Fanuc TP program (LS listing): approach0.LS

/PROG  approach0
/ATTR
OWNER		= MNEDITOR;
COMMENT		= "test_comment";
PROG_SIZE	= 0;
CREATE		= DATE 31-12-14  TIME 12:00:00;
MODIFIED	= DATE 31-12-14  TIME 12:00:00;
FILE_NAME	= ;
VERSION		= 0;
LINE_COUNT	= 2;
MEMORY_SIZE	= 0;
PROTECT		= READ_WRITE;
TCD:  STACK_SIZE	= 0,
      TASK_PRIORITY	= 50,
      TIME_SLICE	= 0,
      BUSY_LAMP_OFF	= 0,
      ABORT_REQUEST	= 0,
      PAUSE_REQUEST	= 0;
DEFAULT_GROUP	= 1,*,*,*,*,*,*;
CONTROL_CODE	= 00000000 00000000;
/MN
   1:L P[1] 100mm/sec FINE ;
   2:L P[2] 101mm/sec FINE ;
/POS
P[1]{
   GP1:
    UF : 9, UT : 9,
	J1=    0.000 deg,	J2=    0.000 deg,	J3=    0.300 deg,
	J4=    0.600 deg,	J5=    0.500 deg,	J6=    10.000 deg,
	E1=  1000.000  mm,	E2=  1000.000  mm
};
P[2]{
   GP1:
    UF : 9, UT : 9,
	J1=    0.000 deg,	J2=    0.000 deg,	J3=    0.000 deg,
	J4=    0.000 deg,	J5=    0.000 deg,	J6=    0.000 deg,
	E1=  1000.000  mm,	E2=  1000.000  mm
};
/END
